Staubli VAL3: init.pgx

public program init()
  local num i
begin
  // setMutex
  setMutex(cycleStatus:bMutex)
  // START CYCLE
  for i=0 to size(saveCycle:nDoneStart)-1
    saveCycle:nDoneStart[i]=0
  endFor
  // PROCESS LIST
  if saveCycle:bLoop
    for i=0 to size(saveCycle:nDoneCycle)-1
      saveCycle:nDoneCycle[i]=0
    endFor
  endIf
  // END CYCLE
  for i=0 to size(saveCycle:nDoneEnd)-1
    saveCycle:nDoneEnd[i]=0
  endFor
  //release
  cycleStatus:bMutex=false
end
